# EPICS substitutions: iocBoot/ioc13GasLoading/remoteControl.substitutions
file "$(CARS)/db/GalilRemoteControl.template"
{
pattern
{    M,         BI0,                BI1}
   {"m7", "Galil1:Galil0Bi0_STATUS", Galil1:Galil0Bi1_STATUS}
   {"m8", "Galil1:Galil0Bi2_STATUS", Galil1:Galil0Bi3_STATUS}
   {"m3", "Galil1:Galil0Bi4_STATUS", Galil1:Galil0Bi5_STATUS}
   {"m4", "Galil1:Galil0Bi6_STATUS", Galil1:Galil0Bi7_STATUS}
   {"m5", "Galil1:Galil1Bi6_STATUS", Galil1:Galil1Bi7_STATUS}
}
